FUNCTION_BLOCK FB_State4 EXTENDS FB_State
VAR_INPUT
END_VAR
VAR_OUTPUT
END_VAR
VAR
END_VAR

END_FUNCTION_BLOCK

(* stored: Version 1.1.0.1, ProductVersion 3.1.4024.12
   POU FB_State4: Id {a7ebef2c-19a5-4130-90b6-f36862d2a4c2}, SpecialFunc None *)
